{attribute 'TcGenerated'}
// This function has been automatically generated from the project information.
VAR_GLOBAL CONSTANT
    {attribute 'const_non_replaced'}
    {attribute 'linkalways'}
    stLibVersion_LFE_VAC : ST_LibVersion := (iMajor := 2, iMinor := 0, iBuild := 1, iRevision := 0, sVersion := '2.0.1');
END_VAR

(* stored: Version 1.1.0.1, ProductVersion 3.1.4022.18
   GVL Global_Version: Id 7cfd6429-9f07-40be-ac2f-f99132ff4f13 *)
